FUNCTION_BLOCK FB_Section_ToolStation IMPLEMENTS I_Section
VAR_INPUT
	bEnable					: BOOL;
END_VAR
VAR_OUTPUT
END_VAR
VAR
	bTriggerToolRotation	: BOOL;
	Modules					: ARRAY [0..2] OF I_Module;	

	fbCoilHolder			: FB_Module_CoilHolder;
	fbToolHolderDoor		: FB_Module_ToolHolderDoor;
	fbToolHolder			: FB_Module_ToolHolder;
	
	idx						: INT;
END_VAR

IF bEnable THEN
	fbCoilHolder(bEnable 			:= TRUE);
	fbToolHolderDoor(bEnable 		:= TRUE);
	fbToolHolder(
			bEnable 				:= TRUE, 
			bToolRotationBtn 		:= bTriggerToolRotation, 
			bToolRotationBtnLight 	:= GVL.bToolingRotationBtnLight);
	
	Modules[0]	:= fbCoilHolder;
	Modules[1]	:= fbToolHolderDoor;
	Modules[2]	:= fbToolHolder;
	
	FOR idx := 0 TO 2 DO
    	Modules[idx].M_Start();
	END_FOR;
	
	IF GVL.bToolingRotationBtn AND fbToolHolderDoor.bDoorUp THEN
		bTriggerToolRotation := TRUE;
	ELSE
		bTriggerToolRotation := FALSE;
	END_IF
END_IF

METHOD M_CloseDoor : BOOL
VAR_INPUT
END_VAR
IF bEnable THEN
	M_CloseDoor := fbToolHolderDoor.M_Up();
END_IF
END_METHOD

METHOD M_Goto : BOOL
VAR_INPUT
	nTargetIndex: INT;
END_VAR

VAR
END_VAR
IF bEnable THEN
	M_Goto := fbCoilHolder.M_GoTo(nTargetIndex := nTargetIndex);
END_IF
END_METHOD

{warning 'add method implementation '}
METHOD M_Halt : BOOL
END_METHOD

METHOD M_OpenDoor : BOOL
VAR_INPUT
END_VAR
IF bEnable THEN
	M_OpenDoor := fbToolHolderDoor.M_Down();
END_IF
END_METHOD

{warning 'add method implementation '}
METHOD M_Start : BOOL
END_METHOD

{warning 'add method implementation '}
METHOD M_Stop : BOOL
END_METHOD

END_FUNCTION_BLOCK

(* stored: Version 1.1.0.1, ProductVersion 3.1.4024.15
   POU FB_Section_ToolStation: Id {511696e8-12f8-47da-a29f-70728d219f59}, SpecialFunc None
   Method M_CloseDoor: Id {14bc3192-cba0-4753-b003-278ffd1c5135}
   Method M_Goto: Id {238912f1-2465-4448-9839-b6a3da1e07f6}
   Method M_Halt: Id {2bdb3e6e-c1a7-478d-95b0-75d93fba08af}
   Method M_OpenDoor: Id {a0c1f1ff-ab52-4f0d-a35e-19942b7a5b42}
   Method M_Start: Id {cabe4c21-79e3-46ea-ba76-d03cb2c651dd}
   Method M_Stop: Id {575e3d9e-84f8-438a-a92f-e2a00552d590} *)
